// TIA Portal project "2022.06.07_Array的用法" (V17)

(* hardware
DEVICE "S7-1200 station_1"  S7-1200 Station
   slot 0: "Rack_0"  S7-1200 Rack  Rack  V1.0
   slot 1: "PLC_1"  CPU 1212C DC/DC/DC  6ES7 212-1AE40-0XB0  V4.5
*)

// ===== PLC "PLC_1"  CPU 1212C DC/DC/DC =====

VAR_GLOBAL   // PLC tag table "默认变量表"
   "模拟量输入" AT %MW100 : Word;
   "Tag_3" AT %MW102 : UInt;
   "Tag_4" AT %MW104 : UInt;
   "Tag_5" AT %MW106 : UInt;
   "Tag_6" AT %I0.0 : Bool;
   "Tag_7" AT %M0.0 : Bool;
   "X(2)" AT %MW10 : Word;
   "Tag_9" AT %MW12 : UInt;
   "X" AT %MW0 : Word;
   "a" AT %MW2 : Word;
   "b" AT %MW4 : Int;
   "c" AT %MW8 : Int;
   "实时温度" AT %MD0 : Real;
   "Tag_10" AT %MD2 : Real;
   "f" AT %MD4 : Real;
   "g" AT %MD8 : Real;
   "X(1)" AT %MD12 : Real;
   "Tag_8" AT %MD16 : Real;
   "中间值(1)" AT %MD200 : Real;
   "中间值" AT %MD104 : Real;
   "工程值" AT %MD108 : Real;
   "要求的频率" AT %MD60 : Real;
   "百分比" AT %MD64 : Real;
   "Tag_12" AT %MW70 : Int;
   "Tag_2" AT %I0.1 : Bool;
   "0" AT %Q0.0 : Bool;
   "加热" AT %Q0.1 : Bool;
END_VAR

DATA_BLOCK "测试数据块_1"   // DB1
{ S7_Optimized_Access := 'FALSE' }
VERSION : 0.1
   VAR
      数组 : Array[0..9] of Bool;
      数组_1 : Array[0..9] of Byte;
      存储器 : DWord;
   END_VAR
BEGIN
END_DATA_BLOCK

ORGANIZATION_BLOCK "Main"   // OB1, LAD, ProgramCycle
TITLE = "Main Program Sweep (Cycle)"
{ S7_Optimized_Access := 'TRUE' }
VERSION : 0.1
   VAR_INPUT
      Initial_Call : Bool;   // Initial call of this OB
      Remanence : Bool;   // =True, if remanent data are available
   END_VAR
BEGIN

REGION Network 1
   // bool开关，字节不能当开关
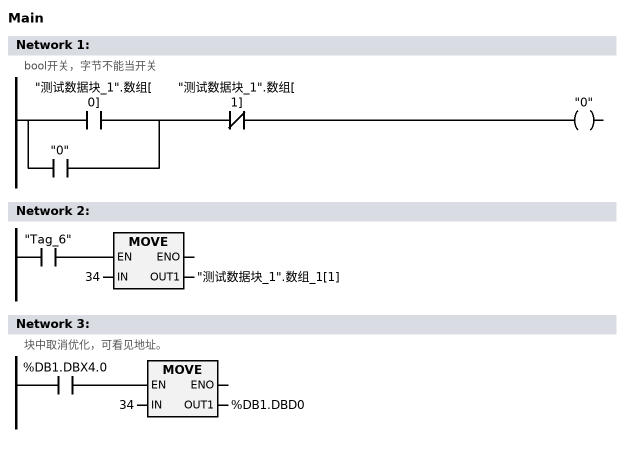
   RUNG wire#powerrail
      Contact( "测试数据块_1".数组[0] )
      wire#w1
      I_Contact( "测试数据块_1".数组[1] )
      Coil( "0" )
   END_RUNG
   RUNG wire#powerrail
      Contact( "0" )
   END_RUNG wire#w1
   // the same network as SCL:
   "0" := ("测试数据块_1".数组[0] OR "0") AND NOT "测试数据块_1".数组[1];
END_REGION

REGION Network 2
   RUNG wire#powerrail
      Contact( "Tag_6" )
      Move(in := 34, out1 => "测试数据块_1".数组_1[1])
   END_RUNG
   // the same network as SCL:
   IF "Tag_6" THEN "测试数据块_1".数组_1[1] := 34; END_IF;
END_REGION

REGION Network 3
   // 块中取消优化，可看见地址。
   RUNG wire#powerrail
      Contact( %DB1.DBX4.0 )
      Move(in := 34, out1 => %DB1.DBD0)
   END_RUNG
   // the same network as SCL:
   IF %DB1.DBX4.0 THEN %DB1.DBD0 := 34; END_IF;
END_REGION
END_ORGANIZATION_BLOCK